FUNCTION_BLOCK Gate
  (* Standard: 61499-2 *)
  (* Version 0,1, 2015-00-15, Th?o, PC_THEO *)
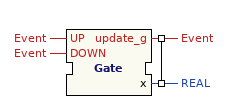
  EVENT_INPUT
    UP;
    DOWN;
  END_EVENT
  EVENT_OUTPUT
    update_g WITH x;
  END_EVENT
  VAR_OUTPUT
    x : REAL;
  END_VAR
  VAR
    C1x : REAL;
    d : REAL;
    k : INT;
  END_VAR
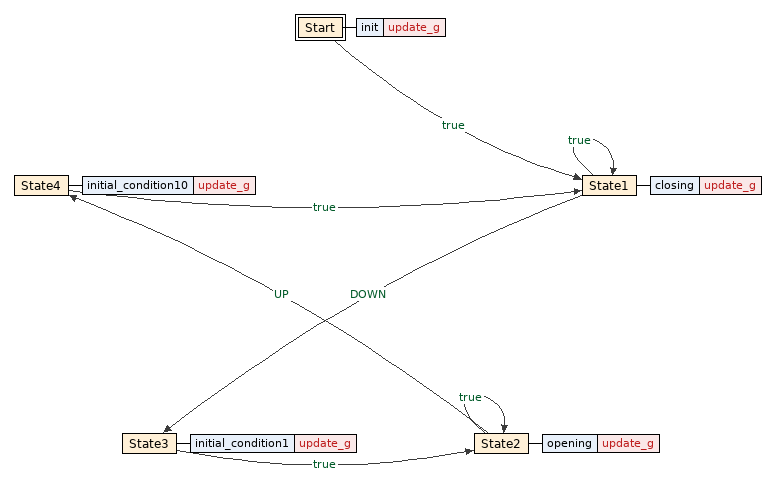
  EC_STATES
    Start : init -> update_g;
    State1 : closing -> update_g;
    State2 : opening -> update_g;
    State3 : initial_condition1 -> update_g;
    State4 : initial_condition10 -> update_g;
  END_STATES
  EC_TRANSITIONS
    Start TO State1 := true;
    State1 TO State3 := DOWN;
    State1 TO State1 := true;
    State2 TO State4 := UP;
    State2 TO State2 := true;
    State3 TO State2 := true;
    State4 TO State1 := true;
  END_TRANSITIONS
  ALGORITHM opening IN C:
me->x = me->C1x*exp(-1.0L/2.0L*me->d*me->k) + 1;
//printf("Gate opening : %f, tick : %d\n", me->x, me->k);
(me->k)++;
  END_ALGORITHM
  ALGORITHM closing IN C:
 me->x = me->C1x*exp(-1.0L/2.0L*me->d*me->k)+10;
 //printf("Gate closing : %f, tick : %d\n", me->x, me->k);
 (me->k)++;
  END_ALGORITHM
  ALGORITHM init IN C:
me->x=10;
me->k=0;
me->d=0.1;
me->C1x=0;
  END_ALGORITHM
  ALGORITHM initial_condition10 IN C:
me->k=0;
me->C1x=me->x-10;
printf("Gate starts opening\n");
  END_ALGORITHM
  ALGORITHM initial_condition1 IN C:
me->k=0;
me->C1x=me->x-1;
printf("Gate starts closing\n");
  END_ALGORITHM
END_FUNCTION_BLOCK
